(* IEC 61131-3 sources: repolevel_ST_code_completion/output/0127完整版本_带planner/repoeval_Builder_Application_RPI/readful_result_before_fix, 5 files *)

(* ---- ConcreteBuilder.st ---- *)
//This is the concrete builder class, reponsible for building the final product object
FUNCTION_BLOCK ConcreteBuilder IMPLEMENTS ITF_Builder
VAR_INPUT
END_VAR
VAR_OUTPUT
END_VAR
VAR
    isCompleted : BOOL := FALSE; // Indicates if the product construction is completed
    isValid : BOOL; // Indicates if the specifications are valid
    i : INT; // Loop variable
END_VAR

// Step 1: Initialize the product object
localProduct := Product();
localProduct.Initialize();

// Step 2: Validate client specifications
isValid := TRUE;
FOR i := 1 TO 4 DO
    IF specifications[i] = '' THEN
        isValid := FALSE;
        EXIT;
    END_IF;
END_FOR;

// Step 3: Update product attributes based on specifications and director guidance
IF isValid THEN
    localProduct.Set_Main_Part(specifications[1]);
    localProduct.Set_Part1(specifications[2]);
    localProduct.Set_Part2(specifications[3]);
    localProduct.Set_Part3(specifications[4]);
END_IF;

// Step 4: Mark product as completed if valid
IF isValid THEN
    isCompleted := TRUE;
    localProduct.Mark_As_Completed();
END_IF;

// Step 5: Return the constructed product object
IF isCompleted THEN
    RETURN localProduct;
ELSE
    RETURN Product(); // Return an empty product if construction failed
END_IF;
END_FUNCTION_BLOCK

(* ---- Director.st ---- *)
{attribute 'enable_dynamic_creation'}
//The director class is responsible to delegate the construction of the final product object
// to a concrete builder object.
FUNCTION_BLOCK Director
VAR_INPUT
	//Reference to the builder that is going to be building the final product object.
	inputConcreteBuilder : ConcreteBuilder(specs := inputConcreteBuilder.specifications);
END_VAR
VAR_OUTPUT
END_VAR
VAR
    product : Product; // Local variable to store the final product object.
END_VAR

IF inputConcreteBuilder <> 0 THEN
    // Assign the input concrete builder to the Director's concreteBuilder field.
    THIS^.concreteBuilder := inputConcreteBuilder;

    // Step-by-step construction of the product using the concrete builder.
    THIS^.concreteBuilder.Set_Main_Part(THIS^.concreteBuilder.specifications[1]);
    THIS^.concreteBuilder.Set_Part1(THIS^.concreteBuilder.specifications[2]);
    THIS^.concreteBuilder.Set_Part2(THIS^.concreteBuilder.specifications[3]);
    THIS^.concreteBuilder.Set_Part3(THIS^.concreteBuilder.specifications[4]);

    // Retrieve the final product object from the concrete builder.
    product := THIS^.concreteBuilder.Get_Result();

    // Return the constructed product object.
    RETURN product;
ELSE
    // If the input concrete builder is invalid, return an empty product object.
    RETURN Product();
END_IF;
END_FUNCTION_BLOCK

(* ---- Product.st ---- *)
{attribute 'enable_dynamic_creation'}
//The class Product is just a plain bluprint of the components of the object to be built.
//The final Product may ot may not contain the all the Parts listed on the Product declaration
// rather only the parts in the specifications sent by the client.
FUNCTION_BLOCK Product
VAR_INPUT
	//List of possible parts to be build in a final Product object
	mainPart 	: STRING;
	part1 		: STRING;
	part2 		: STRING;
	part3 		: STRING;
END_VAR
VAR_OUTPUT
END_VAR
VAR
    selectedParts : ARRAY [1..4] OF STRING := ['', '', '', ''];
    index         : INT := 1;
END_VAR

IF mainPart <> '' THEN
    selectedParts[index] := mainPart;
    index := index + 1;
END_IF;

IF part1 <> '' THEN
    selectedParts[index] := part1;
    index := index + 1;
END_IF;

IF part2 <> '' THEN
    selectedParts[index] := part2;
    index := index + 1;
END_IF;

IF part3 <> '' THEN
    selectedParts[index] := part3;
    index := index + 1;
END_IF;

localProduct.mainPart := selectedParts[1];
localProduct.part1 := selectedParts[2];
localProduct.part2 := selectedParts[3];
localProduct.part3 := selectedParts[4];
END_FUNCTION_BLOCK

(* ---- Director_Construct.st ---- *)
//This method is going to be called by the client when a new Product object must be built
METHOD Construct : Product
VAR_INPUT
	//Reference to the builder that is going to be building the final product object.
	inputConcreteBuilder : ConcreteBuilder(specs := inputConcreteBuilder.specifications);
END_VAR
VAR_OUTPUT
END_VAR
VAR
    specifications : ARRAY [1..4] OF STRING;
    finalProduct : Product;
END_VAR

// Step 1: Retrieve specifications from inputConcreteBuilder
specifications := inputConcreteBuilder.specifications;

// Step 2: Initialize a new Product object using inputConcreteBuilder
inputConcreteBuilder.Initialize_Product();

// Step 3: Build the Product step by step based on specifications
inputConcreteBuilder.Set_Main_Part(specifications[1]);
inputConcreteBuilder.Set_Part1(specifications[2]);
inputConcreteBuilder.Set_Part2(specifications[3]);
inputConcreteBuilder.Set_Part3(specifications[4]);

// Step 4: Confirm Product construction is complete and return the final Product
finalProduct := inputConcreteBuilder.Get_Result();
Construct := finalProduct;
RETURN;
END_OTHER

(* ---- Product_toString.st ---- *)
//Method to be used in the visualization element for an easier String handling
METHOD toString : STRING
VAR_INPUT
	//List of possible parts to be build in a final Product object
	mainPart 	: STRING;
	part1 		: STRING;
	part2 		: STRING;
	part3 		: STRING;
END_VAR
VAR_OUTPUT
END_VAR
VAR
    tempString : STRING := ''; // Initialize an empty string for the final result
END_VAR

IF mainPart <> '' THEN
    tempString := CONCAT(tempString, mainPart); // Add mainPart if not empty
END_IF;

IF part1 <> '' THEN
    tempString := CONCAT(tempString, part1); // Add part1 if not empty
END_IF;

IF part2 <> '' THEN
    tempString := CONCAT(tempString, part2); // Add part2 if not empty
END_IF;

IF part3 <> '' THEN
    tempString := CONCAT(tempString, part3); // Add part3 if not empty
END_IF;

toString := tempString; // Return the concatenated result
END_OTHER
